Fanuc KAREL source: JOINT2POS.kl

PROGRAM T
%NOLOCKGROUP
VAR
 v0 : JOINTPOS
 v1 : POSITION
 v2 : POSITION
 v3 : INTEGER
 v4 : POSITION
 v5 : CONFIG
 v6 : ARRAY[6] OF REAL
 v7 : INTEGER
BEGIN
 JOINT2POS(v0, v1, v2, v3, v4, v5, v6, v7)
END T
